TYPE ST_Point :
STRUCT
	x : INT;
	y : INT;
END_STRUCT
END_TYPE

(* stored: Version 1.1.0.1, ProductVersion 3.1.4024.12
   POU ST_Point: Id {dfcc0369-15ad-48aa-8c88-2294f0f643cf}, SpecialFunc None *)
